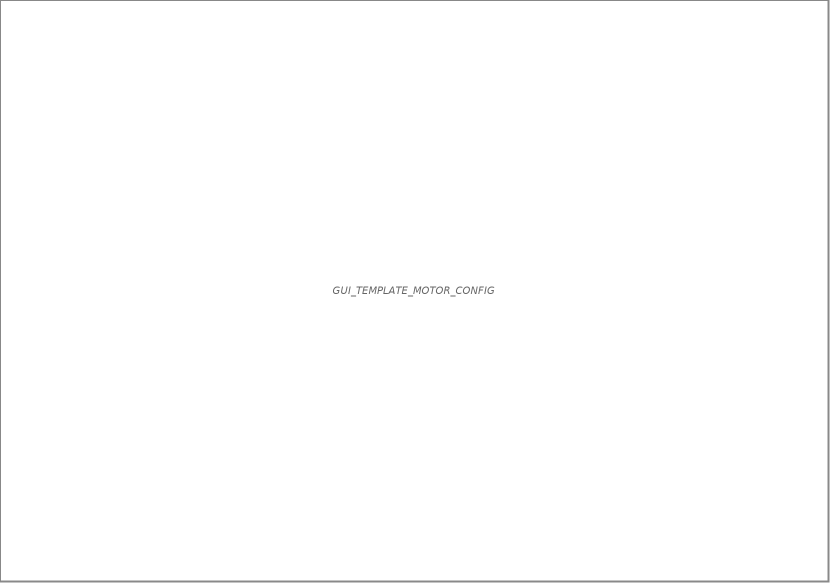
VISUALIZATION GUI_Motor002_Cfg  // 830x583
    Frame (0,0 828x581)
        shows GUI_TEMPLATE_MOTOR_CONFIG(m_Instance := MAIN.Motor002)
END_VISUALIZATION

(* stored: Version 1.1.0.1, ProductVersion 3.1.4024.3
   Visu GUI_Motor002_Cfg: Id {3a1ef2e8-5f92-4e54-afbb-c0ded10dd311} *)
